Fanuc KAREL source: kb00106.KL

-- PROVISIONAL review KL for V770-1; original PC SHA256 91f27d2d2201b27b1e33a9115a21ebeaba31023dfd0077e3b9f1d05da0483514
-- Incomplete behavior may be omitted. Consult companion uncertainty JSON. Do not deploy.
PROGRAM KB00106
%NOLOCKGROUP
BEGIN
  -- UNRESOLVED_PC offsets 5-15; opcodes 27,22,31
  -- UNRESOLVED_PC offsets 20-24; opcodes 7F
END KB00106
